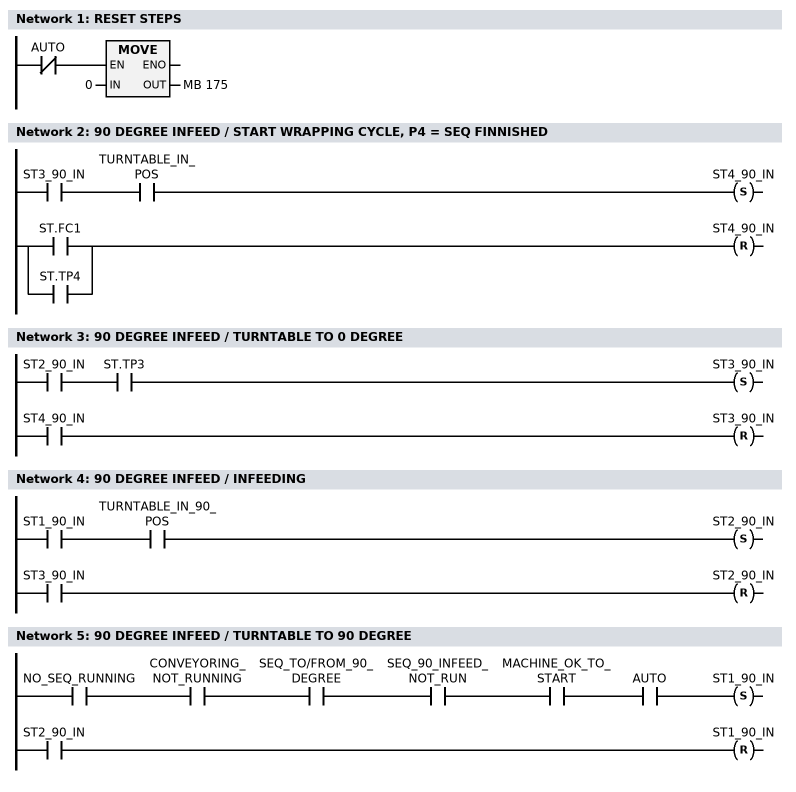
[picture p24: 90_DEGREE_INFEED networks 1-5]
NETWORK
TITLE = RESET STEPS
      AN    "AUTO";
      JNB   _001;
      L     0;
      T     MB 175;
_001: NOP   0;
NETWORK
TITLE = 90 DEGREE INFEED / START WRAPPING CYCLE, P4 = SEQ FINNISHED
      A     "ST3_90_IN";
      A     "TURNTABLE_IN_POS";
      S     "ST4_90_IN";
      A(;
      O     "ST.FC1";
      O     "ST.TP4";
      );
      R     "ST4_90_IN";
      NOP   0;
NETWORK
TITLE = 90 DEGREE INFEED / TURNTABLE TO 0 DEGREE
      A     "ST2_90_IN";
      A     "ST.TP3";
      S     "ST3_90_IN";
      A     "ST4_90_IN";
      R     "ST3_90_IN";
      NOP   0;
NETWORK
TITLE = 90 DEGREE INFEED / INFEEDING
      A     "ST1_90_IN";
      A     "TURNTABLE_IN_90_POS";
      S     "ST2_90_IN";
      A     "ST3_90_IN";
      R     "ST2_90_IN";
      NOP   0;
NETWORK
TITLE = 90 DEGREE INFEED / TURNTABLE TO 90 DEGREE
      A     "NO_SEQ_RUNNING";
      A     "CONVEYORING_NOT_RUNNING";
      A     "SEQ_TO/FROM_90_DEGREE";
      A     "SEQ_90_INFEED_NOT_RUN";
      A     "MACHINE_OK_TO_START";
      A     "AUTO";
      S     "ST1_90_IN";
      A     "ST2_90_IN";
      R     "ST1_90_IN";
      NOP   0;
END_FUNCTION

FUNCTION "90_DEGREE_OUTFEED" : VOID	// FC 18
TITLE = 90 DEGREE OUTFEED, OPTION
AUTHOR : LKA
NAME : OUTF_90D
VERSION : 0.1
BEGIN
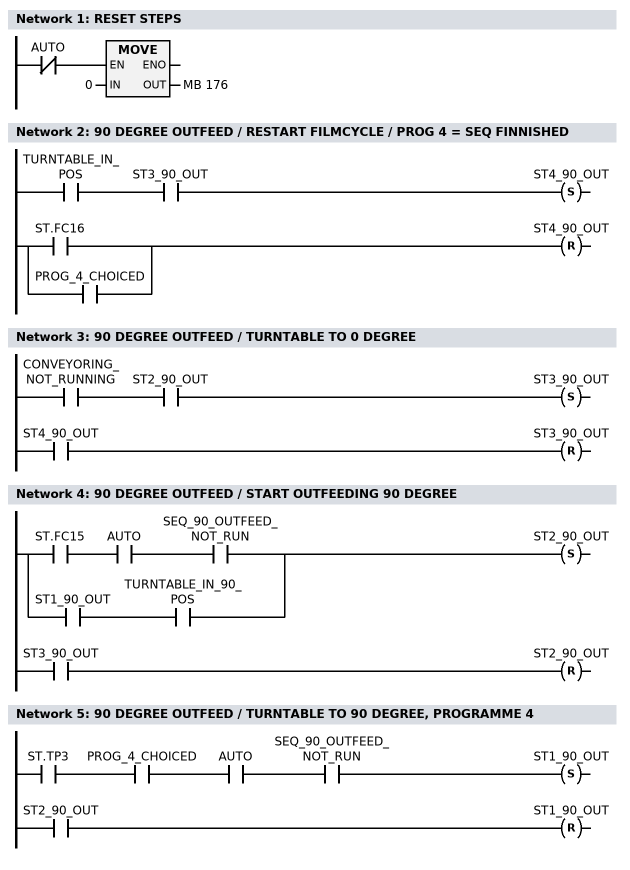
NETWORK
TITLE = RESET STEPS
      AN    "AUTO";
      JNB   _001;
      L     0;
      T     MB 176;
_001: NOP   0;
NETWORK
TITLE = 90 DEGREE OUTFEED / RESTART FILMCYCLE / PROG 4 = SEQ FINNISHED
      A     "TURNTABLE_IN_POS";
      A     "ST3_90_OUT";
      S     "ST4_90_OUT";
      A(;
      O     "ST.FC16";
      O     "PROG_4_CHOICED";
      );
      R     "ST4_90_OUT";
      NOP   0;
NETWORK
TITLE = 90 DEGREE OUTFEED / TURNTABLE TO 0 DEGREE
      A     "CONVEYORING_NOT_RUNNING";
      A     "ST2_90_OUT";
      S     "ST3_90_OUT";
      A     "ST4_90_OUT";
      R     "ST3_90_OUT";
      NOP   0;
NETWORK
TITLE = 90 DEGREE OUTFEED / START OUTFEEDING 90 DEGREE
      A(;
      A     "ST.FC15";
      A     "AUTO";
      A     "SEQ_90_OUTFEED_NOT_RUN";
      O;
      A     "ST1_90_OUT";
      A     "TURNTABLE_IN_90_POS";
      );
      S     "ST2_90_OUT";
      A     "ST3_90_OUT";
      R     "ST2_90_OUT";
      NOP   0;
NETWORK
TITLE = 90 DEGREE OUTFEED / TURNTABLE TO 90 DEGREE, PROGRAMME 4
      A     "ST.TP3";
      A     "PROG_4_CHOICED";
      A     "AUTO";
      A     "SEQ_90_OUTFEED_NOT_RUN";
      S     "ST1_90_OUT";
      A     "ST2_90_OUT";
      R     "ST1_90_OUT";
      NOP   0;
END_FUNCTION

FUNCTION "TURN_TO/FROM_90_DEG" : VOID	// FC 19
TITLE = TURNTABLE TO OR FROM 90 DEGREE, OPTION
AUTHOR : LKA
NAME : TT_90
VERSION : 0.1
BEGIN
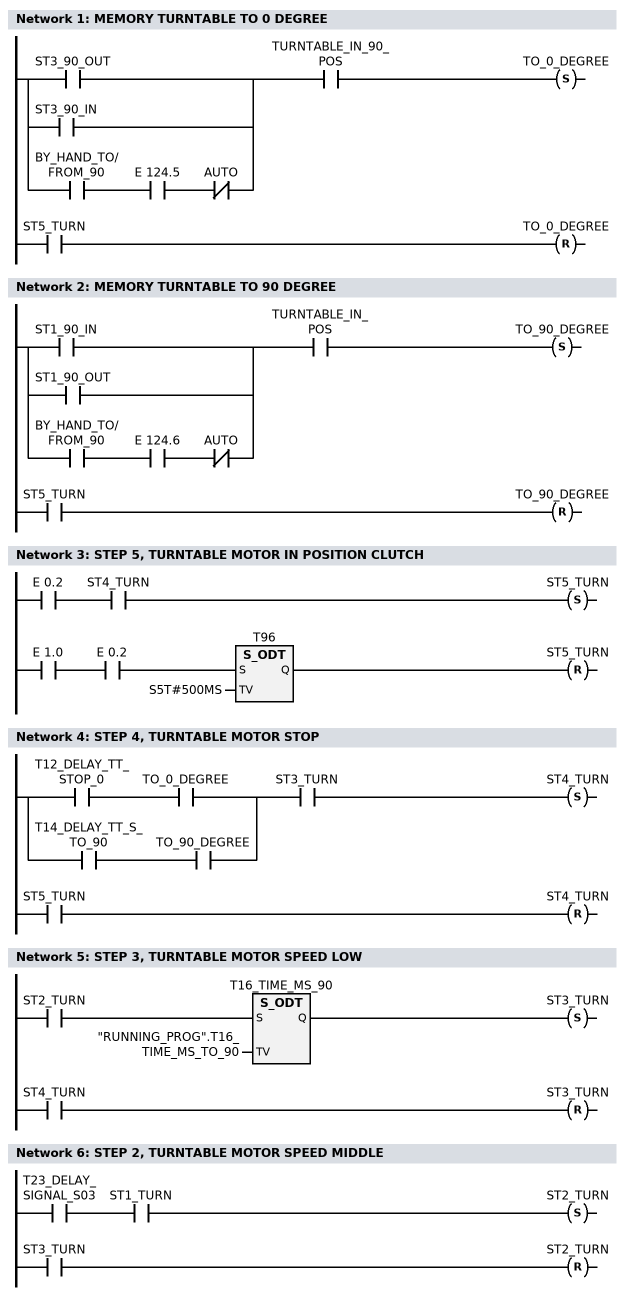
NETWORK
TITLE = MEMORY TURNTABLE TO 0 DEGREE
      A(;
      O     "ST3_90_OUT";
      O     "ST3_90_IN";
      O;
      A     "BY_HAND_TO/FROM_90";
      A     "E 124.5";
      AN    "AUTO";
      );
      A     "TURNTABLE_IN_90_POS";
      S     "TO_0_DEGREE";
      A     "ST5_TURN";
      R     "TO_0_DEGREE";
      NOP   0;
NETWORK
TITLE = MEMORY TURNTABLE TO 90 DEGREE
      A(;
      O     "ST1_90_IN";
      O     "ST1_90_OUT";
      O;
      A     "BY_HAND_TO/FROM_90";
      A     "E 124.6";
      AN    "AUTO";
      );
      A     "TURNTABLE_IN_POS";
      S     "TO_90_DEGREE";
      A     "ST5_TURN";
      R     "TO_90_DEGREE";
      NOP   0;
NETWORK
TITLE = STEP 5, TURNTABLE MOTOR IN POSITION CLUTCH
      A     "E 0.2";
      A     "ST4_TURN";
      S     "ST5_TURN";
      A     "E 1.0";
      A(;
      A     "E 0.2";
      L     S5T#500MS;
      SD    "T96";
      NOP   0;
      NOP   0;
      NOP   0;
      A     "T96";
      );
      R     "ST5_TURN";
      NOP   0;
NETWORK
TITLE = STEP 4, TURNTABLE MOTOR STOP
      A(;
      A     "T12_DELAY_TT_STOP_0";
      A     "TO_0_DEGREE";
      O;
      A     "T14_DELAY_TT_S_TO_90";
      A     "TO_90_DEGREE";
      );
      A     "ST3_TURN";
      S     "ST4_TURN";
      A     "ST5_TURN";
      R     "ST4_TURN";
      NOP   0;
NETWORK
TITLE = STEP 3, TURNTABLE MOTOR SPEED LOW
      A(;
      A     "ST2_TURN";
      L     "RUNNING_PROG".T16_TIME_MS_TO_90;
      SD    "T16_TIME_MS_90";
      NOP   0;
      NOP   0;
      NOP   0;
      A     "T16_TIME_MS_90";
      );
      S     "ST3_TURN";
      A     "ST4_TURN";
      R     "ST3_TURN";
      NOP   0;
NETWORK
TITLE = STEP 2, TURNTABLE MOTOR SPEED MIDDLE
      A     "T23_DELAY_SIGNAL_S03";
      A     "ST1_TURN";
      S     "ST2_TURN";
      A     "ST3_TURN";
      R     "ST2_TURN";
      NOP   0;
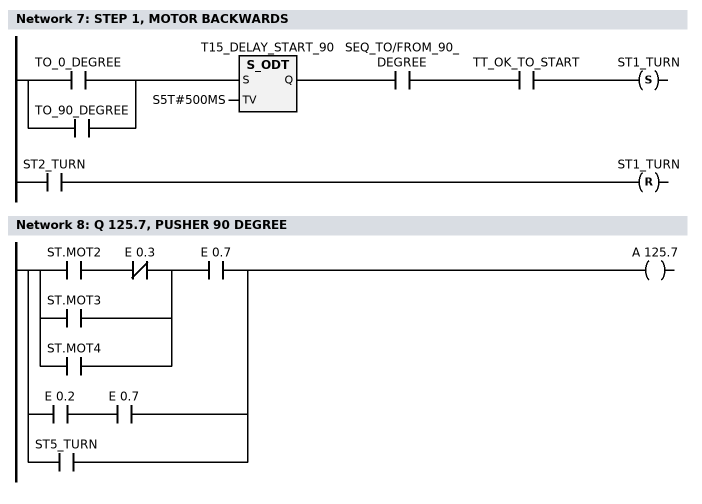
NETWORK
TITLE = STEP 1, MOTOR BACKWARDS
      A(;
      A(;
      O     "TO_0_DEGREE";
      O     "TO_90_DEGREE";
      );
      L     S5T#500MS;
      SD    "T15_DELAY_START_90";
      NOP   0;
      NOP   0;
      NOP   0;
      A     "T15_DELAY_START_90";
      );
      A     "SEQ_TO/FROM_90_DEGREE";
      A     "TT_OK_TO_START";
      S     "ST1_TURN";
      A     "ST2_TURN";
      R     "ST1_TURN";
      NOP   0;
NETWORK
TITLE = Q 125.7, PUSHER 90 DEGREE
      A(;
      A     "ST.MOT2";
      AN    "E 0.3";
      O     "ST.MOT3";
      O     "ST.MOT4";
      );
      A     "E 0.7";
      O;
      A     "E 0.2";
      A     "E 0.7";
      O     "ST5_TURN";
      =     "A 125.7";
END_FUNCTION

FUNCTION "PALLET_POS" : VOID	// FC 21
TITLE = PALLET POSITION - LENGTH MEASURING, OPTION
//OPTIMIZATION OF PALLET STOPTIME ON TURNTABLE
//
//STEP 1: ADJUST CONVEYOR HEIGHT TO BE EQUAL TO STRETCHWRAPPER CONVEYOR, USE A 
//LONG BUBBLE LEVEL.
//
//STEP 2: ADJUST CONVEYOR SPEED ON STRETCHWRAPPER TO BE EQUAL TO INFEEDING 
//CONVEYOR, CHANGE VALUE ON OP3, "TABLEPARAMETERS / CONVEYOR SPEED"
//
//STEP 3: INFEED THE LONGEST PALLET, LOOK AT THE STOP POSITION. ADJUST "Length 
//measuring value" ON OP3 UNTIL THE PALLET STANDS IN MIDDLE. (Counter)
//
//(IF PALLET STOPS TO LATE INCREASE VALUE)
//
//STEP 4: IF NECESSARY, ADJUST OFF DELAY TIME VALUE, T51 & T53 FILTER TIME TO MAKE
//SIGNAL STABLE. (TO LONG TIME MAY CREATE PROBLEM)
AUTHOR : LKA
NAME : L_MATN
VERSION : 1.0
BEGIN
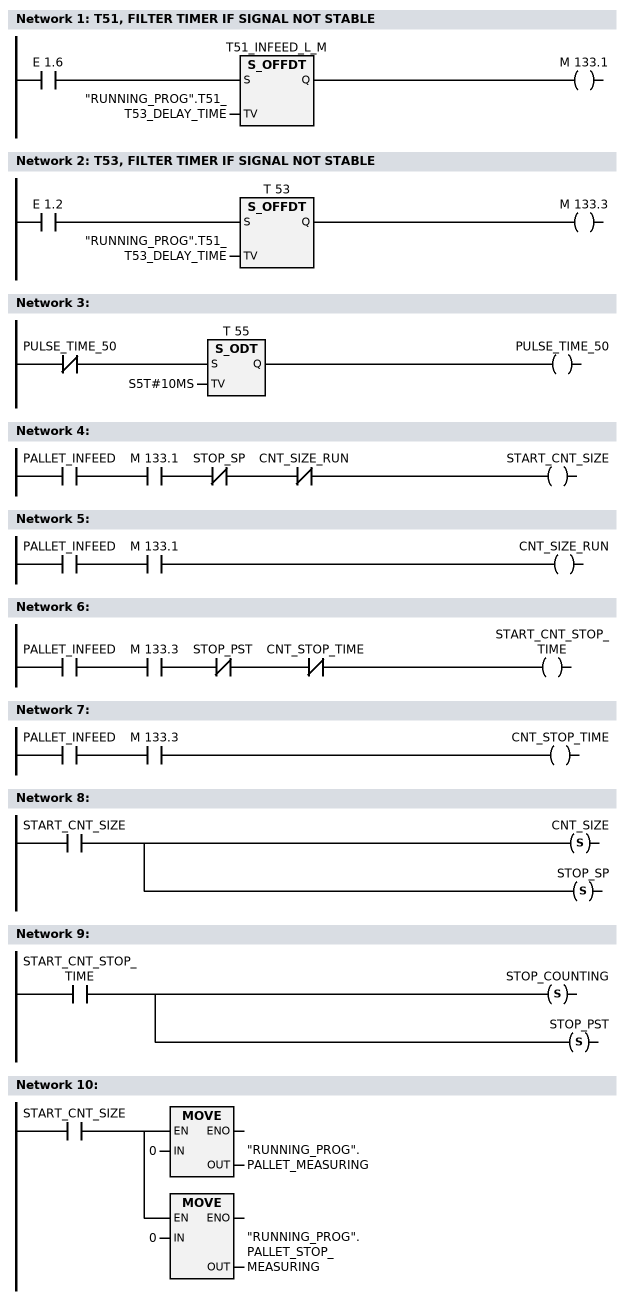
NETWORK
TITLE = T51, FILTER TIMER IF SIGNAL NOT STABLE
      A     "E 1.6";
      L     "RUNNING_PROG".T51_T53_DELAY_TIME;
      SF    "T51_INFEED_L_M";
      NOP   0;
      NOP   0;
      NOP   0;
      A     "T51_INFEED_L_M";
      =     M 133.1;
NETWORK
TITLE = T53, FILTER TIMER IF SIGNAL NOT STABLE
      A     "E 1.2";
      L     "RUNNING_PROG".T51_T53_DELAY_TIME;
      SF    T 53;
      NOP   0;
      NOP   0;
      NOP   0;
      A     T 53;
      =     M 133.3;
NETWORK
TITLE =
      AN    "PULSE_TIME_50";
      L     S5T#10MS;
      SD    T 55;
      NOP   0;
      NOP   0;
      NOP   0;
      A     T 55;
      =     "PULSE_TIME_50";
NETWORK
TITLE =
      A     "PALLET_INFEED";
      A     M 133.1;
      AN    "STOP_SP";
      AN    "CNT_SIZE_RUN";
      =     "START_CNT_SIZE";
NETWORK
TITLE =
      A     "PALLET_INFEED";
      A     M 133.1;
      =     "CNT_SIZE_RUN";
NETWORK
TITLE =
      A     "PALLET_INFEED";
      A     M 133.3;
      AN    "STOP_PST";
      AN    "CNT_STOP_TIME";
      =     "START_CNT_STOP_TIME";
NETWORK
TITLE =
      A     "PALLET_INFEED";
      A     M 133.3;
      =     "CNT_STOP_TIME";
NETWORK
TITLE =
      A     "START_CNT_SIZE";
      S     "CNT_SIZE";
      S     "STOP_SP";
NETWORK
TITLE =
      A     "START_CNT_STOP_TIME";
      S     "STOP_COUNTING";
      S     "STOP_PST";
NETWORK
TITLE =
      A     "START_CNT_SIZE";
      =     L 172.0;
      A     L 172.0;
      JNB   _001;
      L     0;
      T     "RUNNING_PROG".PALLET_MEASURING;
_001: NOP   0;
      A     L 172.0;
      JNB   _002;
      L     0;
      T     "RUNNING_PROG".PALLET_STOP_MEASURING;
_002: NOP   0;
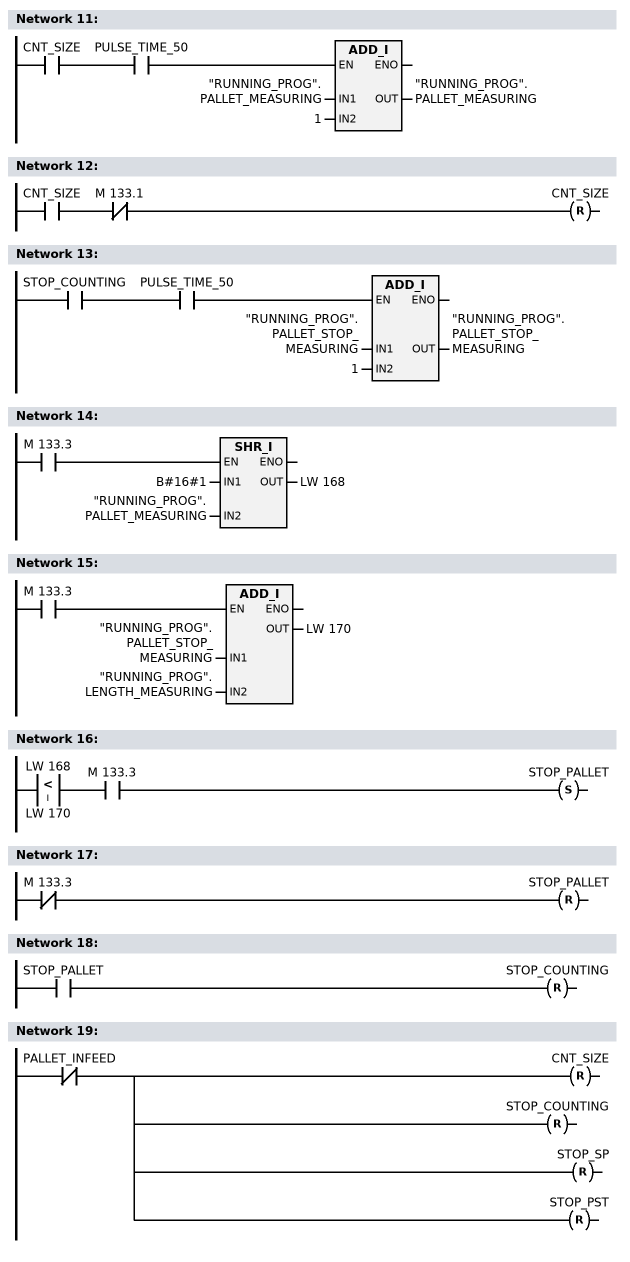
NETWORK
TITLE =
      A     "CNT_SIZE";
      A     "PULSE_TIME_50";
      JNB   _003;
      L     "RUNNING_PROG".PALLET_MEASURING;
      L     1;
      +I;
      T     "RUNNING_PROG".PALLET_MEASURING;
_003: NOP   0;
NETWORK
TITLE =
      A     "CNT_SIZE";
      AN    M 133.1;
      R     "CNT_SIZE";
NETWORK
TITLE =
      A     "STOP_COUNTING";
      A     "PULSE_TIME_50";
      JNB   _004;
      L     "RUNNING_PROG".PALLET_STOP_MEASURING;
      L     1;
      +I;
      T     "RUNNING_PROG".PALLET_STOP_MEASURING;
_004: NOP   0;
NETWORK
TITLE =
      A     M 133.3;
      JNB   _005;
      L     B#16#1;
      L     "RUNNING_PROG".PALLET_MEASURING;
      SSI;
      T     LW 168;
_005: NOP   0;
NETWORK
TITLE =
      A     M 133.3;
      JNB   _006;
      L     "RUNNING_PROG".PALLET_STOP_MEASURING;
      L     "RUNNING_PROG".LENGTH_MEASURING;
      +I;
      T     LW 170;
_006: NOP   0;
NETWORK
TITLE =
      A(;
      L     LW 168;
      L     LW 170;
      <I;
      );
      A     M 133.3;
      S     "STOP_PALLET";
NETWORK
TITLE =
      AN    M 133.3;
      R     "STOP_PALLET";
NETWORK
TITLE =
      A     "STOP_PALLET";
      R     "STOP_COUNTING";
NETWORK
TITLE =
      AN    "PALLET_INFEED";
      R     "CNT_SIZE";
      R     "STOP_COUNTING";
      R     "STOP_SP";
      R     "STOP_PST";
END_FUNCTION

FUNCTION "TURNTABLE" : VOID	// FC 22
TITLE = TURNTABLE
AUTHOR : LKA
NAME : TURNTAB
VERSION : 0.0
BEGIN
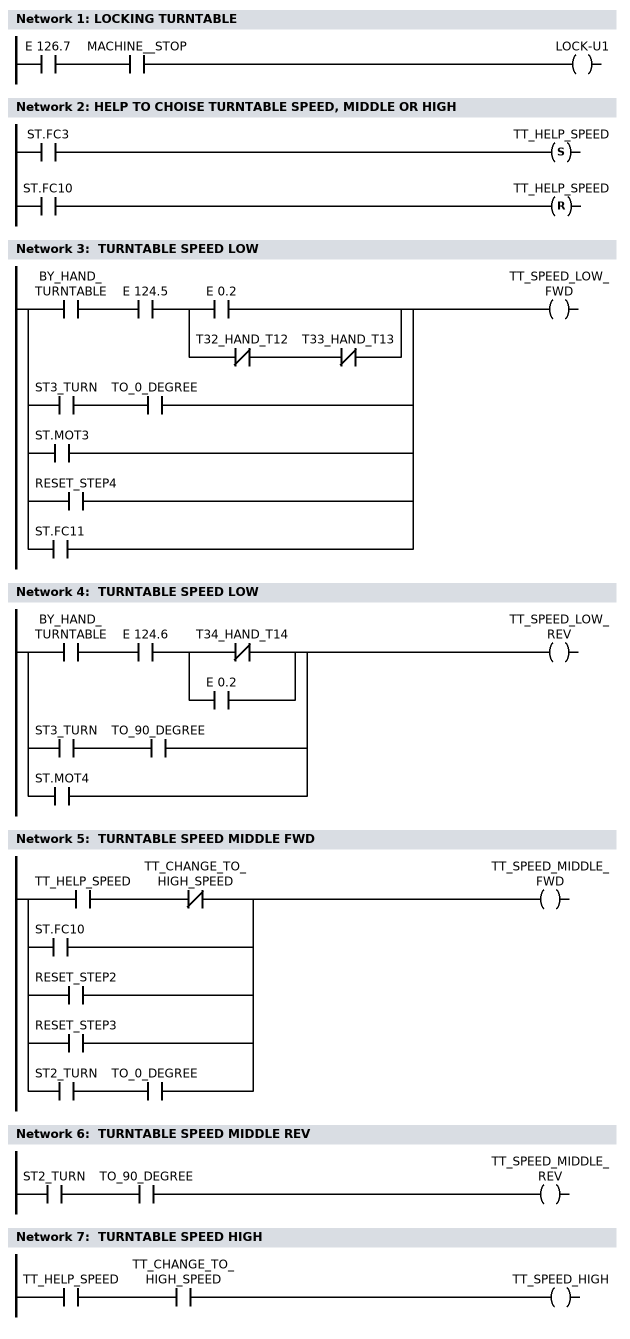
NETWORK
TITLE = LOCKING TURNTABLE
      A     "E 126.7";
      A     "MACHINE__STOP";
      =     "LOCK-U1";
NETWORK
TITLE = HELP TO CHOISE TURNTABLE SPEED, MIDDLE OR HIGH
      A     "ST.FC3";
      S     "TT_HELP_SPEED";
      A     "ST.FC10";
      R     "TT_HELP_SPEED";
      NOP   0;
NETWORK
TITLE =  TURNTABLE SPEED LOW
      A     "BY_HAND_TURNTABLE";
      A     "E 124.5";
      A(;
      O     "E 0.2";
      O;
      AN    "T32_HAND_T12";
      AN    "T33_HAND_T13";
      );
      O;
      A     "ST3_TURN";
      A     "TO_0_DEGREE";
      O     "ST.MOT3";
      O     "RESET_STEP4";
      O     "ST.FC11";
      =     "TT_SPEED_LOW_FWD";
NETWORK
TITLE =  TURNTABLE SPEED LOW
      A     "BY_HAND_TURNTABLE";
      A     "E 124.6";
      A(;
      ON    "T34_HAND_T14";
      O     "E 0.2";
      );
      O;
      A     "ST3_TURN";
      A     "TO_90_DEGREE";
      O     "ST.MOT4";
      =     "TT_SPEED_LOW_REV";
NETWORK
TITLE =  TURNTABLE SPEED MIDDLE FWD
      A     "TT_HELP_SPEED";
      AN    "TT_CHANGE_TO_HIGH_SPEED";
      O     "ST.FC10";
      O     "RESET_STEP2";
      O     "RESET_STEP3";
      O;
      A     "ST2_TURN";
      A     "TO_0_DEGREE";
      =     "TT_SPEED_MIDDLE_FWD";
NETWORK
TITLE =  TURNTABLE SPEED MIDDLE REV
      A     "ST2_TURN";
      A     "TO_90_DEGREE";
      =     "TT_SPEED_MIDDLE_REV";
NETWORK
TITLE =  TURNTABLE SPEED HIGH
      A     "TT_HELP_SPEED";
      A     "TT_CHANGE_TO_HIGH_SPEED";
      =     "TT_SPEED_HIGH";
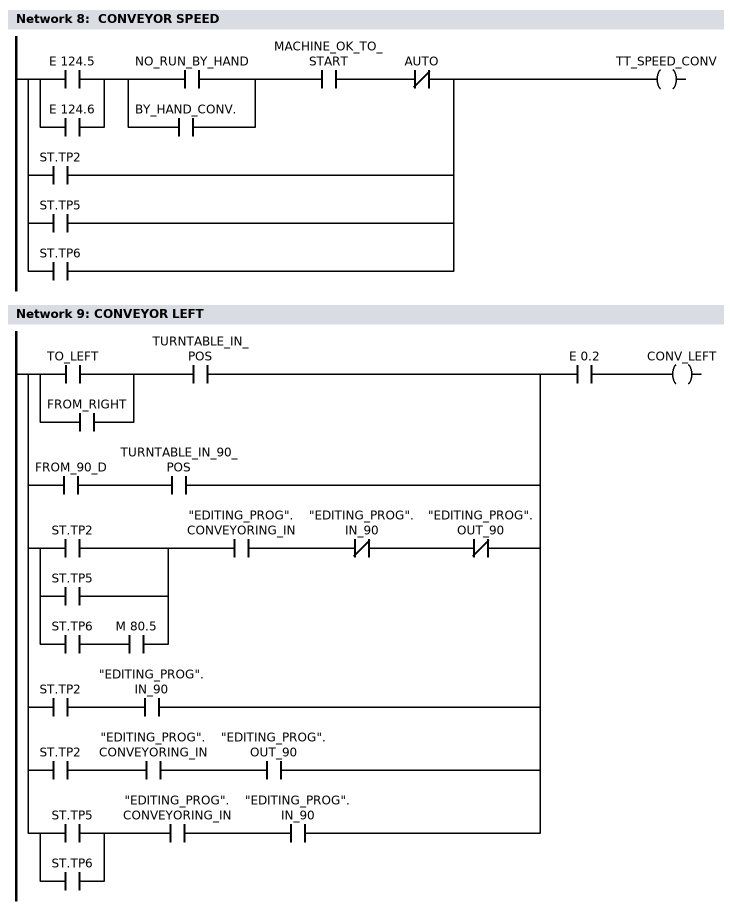
NETWORK
TITLE =  CONVEYOR SPEED
      A(;
      O     "E 124.5";
      O     "E 124.6";
      );
      A(;
      O     "NO_RUN_BY_HAND";
      O     "BY_HAND_CONV.";
      );
      A     "MACHINE_OK_TO_START";
      AN    "AUTO";
      O     "ST.TP2";
      O     "ST.TP5";
      O     "ST.TP6";
      =     "TT_SPEED_CONV";
NETWORK
TITLE = CONVEYOR LEFT
      A(;
      A(;
      O     "TO_LEFT";
      O     "FROM_RIGHT";
      );
      A     "TURNTABLE_IN_POS";
      O;
      A     "FROM_90_D";
      A     "TURNTABLE_IN_90_POS";
      O;
      A(;
      O     "ST.TP2";
      O     "ST.TP5";
      O;
      A     "ST.TP6";
      A     "M 80.5";
      );
      A     "EDITING_PROG".CONVEYORING_IN;
      AN    "EDITING_PROG".IN_90;
      AN    "EDITING_PROG".OUT_90;
      O;
      A     "ST.TP2";
      A     "EDITING_PROG".IN_90;
      O;
      A     "ST.TP2";
      A     "EDITING_PROG".CONVEYORING_IN;
      A     "EDITING_PROG".OUT_90;
      O;
      A(;
      O     "ST.TP5";
      O     "ST.TP6";
      );
      A     "EDITING_PROG".CONVEYORING_IN;
      A     "EDITING_PROG".IN_90;
      );
      A     "E 0.2";
      =     "CONV_LEFT";
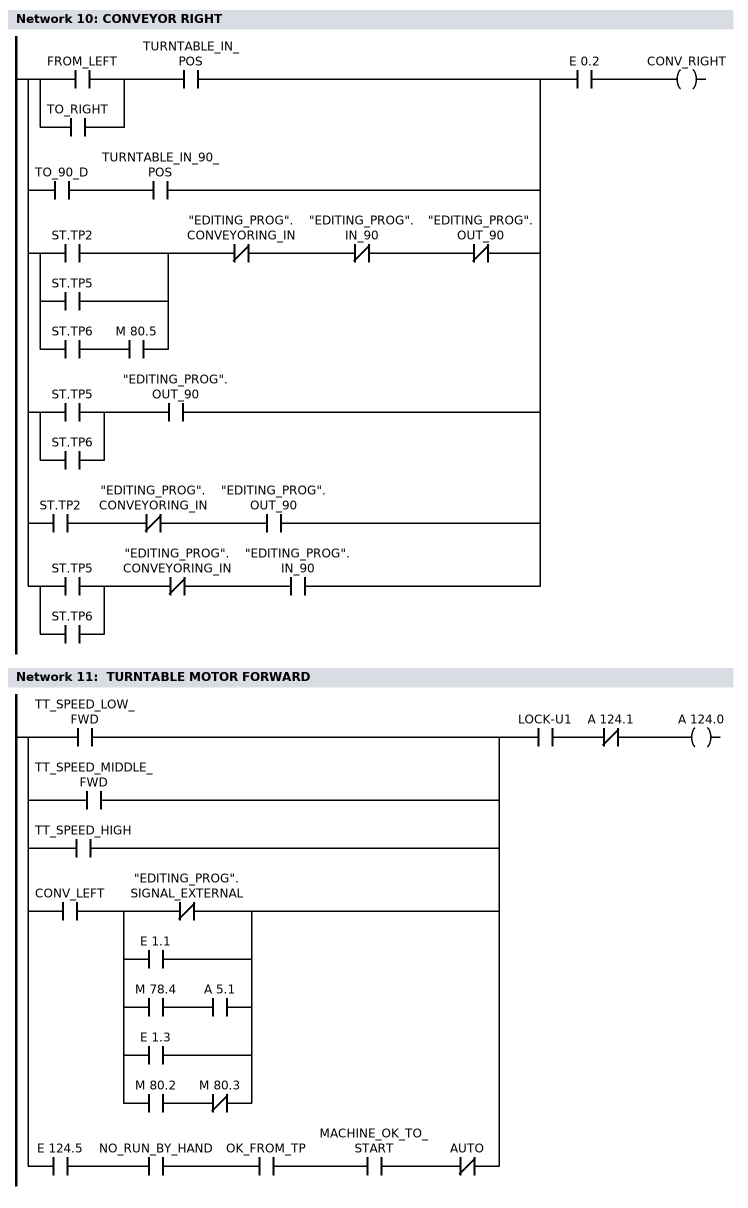
NETWORK
TITLE = CONVEYOR RIGHT
      A(;
      A(;
      O     "FROM_LEFT";
      O     "TO_RIGHT";
      );
      A     "TURNTABLE_IN_POS";
      O;
      A     "TO_90_D";
      A     "TURNTABLE_IN_90_POS";
      O;
      A(;
      O     "ST.TP2";
      O     "ST.TP5";
      O;
      A     "ST.TP6";
      A     "M 80.5";
      );
      AN    "EDITING_PROG".CONVEYORING_IN;
      AN    "EDITING_PROG".IN_90;
      AN    "EDITING_PROG".OUT_90;
      O;
      A(;
      O     "ST.TP5";
      O     "ST.TP6";
      );
      A     "EDITING_PROG".OUT_90;
      O;
      A     "ST.TP2";
      AN    "EDITING_PROG".CONVEYORING_IN;
      A     "EDITING_PROG".OUT_90;
      O;
      A(;
      O     "ST.TP5";
      O     "ST.TP6";
      );
      AN    "EDITING_PROG".CONVEYORING_IN;
      A     "EDITING_PROG".IN_90;
      );
      A     "E 0.2";
      =     "CONV_RIGHT";
NETWORK
TITLE =  TURNTABLE MOTOR FORWARD
      A(;
      O     "TT_SPEED_LOW_FWD";
      O     "TT_SPEED_MIDDLE_FWD";
      O     "TT_SPEED_HIGH";
      O;
      A     "CONV_LEFT";
      A(;
      ON    "EDITING_PROG".SIGNAL_EXTERNAL;
      O     "E 1.1";
      O;
      A     "M 78.4";
      A     "A 5.1";
      O     "E 1.3";
      O;
      A     "M 80.2";
      AN    "M 80.3";
      );
      O;
      A     "E 124.5";
      A     "NO_RUN_BY_HAND";
      A     "OK_FROM_TP";
      A     "MACHINE_OK_TO_START";
      AN    "AUTO";
      );
      A     "LOCK-U1";
      AN    "A 124.1";
      =     "A 124.0";
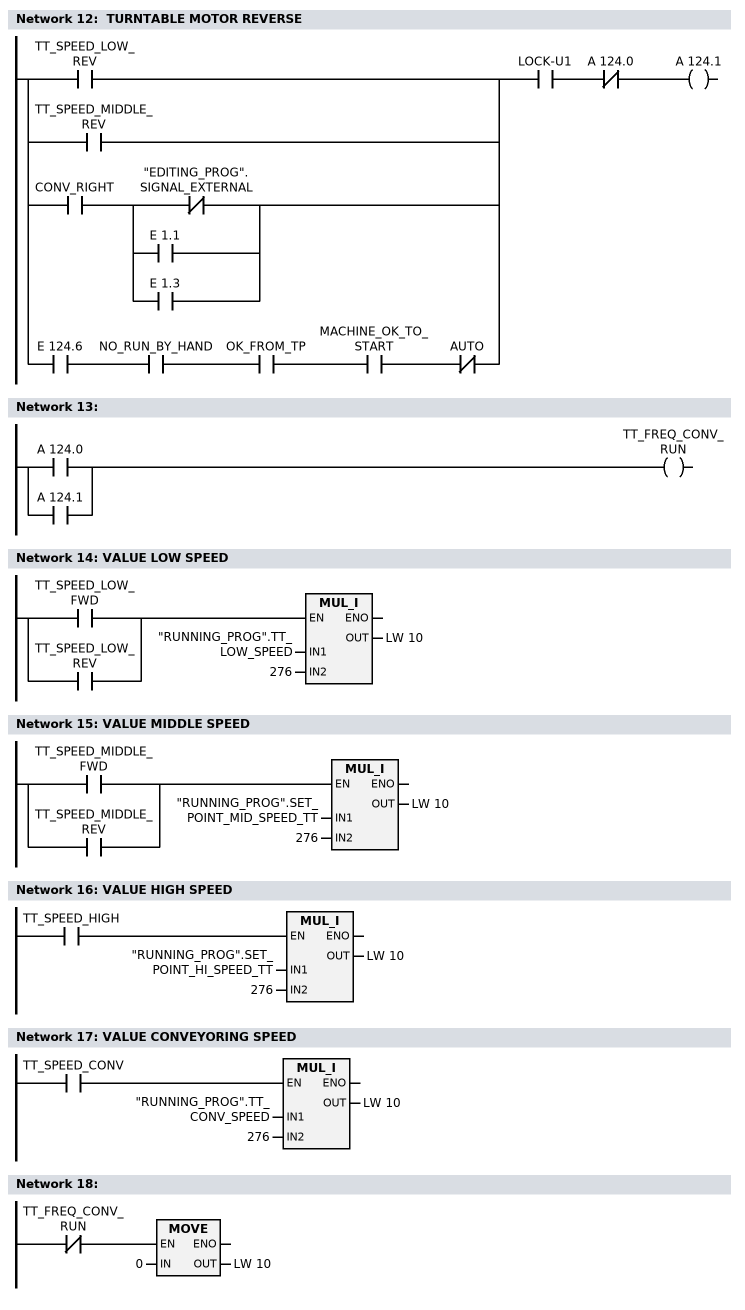
NETWORK
TITLE =  TURNTABLE MOTOR REVERSE
      A(;
      O     "TT_SPEED_LOW_REV";
      O     "TT_SPEED_MIDDLE_REV";
      O;
      A     "CONV_RIGHT";
      A(;
      ON    "EDITING_PROG".SIGNAL_EXTERNAL;
      O     "E 1.1";
      O     "E 1.3";
      );
      O;
      A     "E 124.6";
      A     "NO_RUN_BY_HAND";
      A     "OK_FROM_TP";
      A     "MACHINE_OK_TO_START";
      AN    "AUTO";
      );
      A     "LOCK-U1";
      AN    "A 124.0";
      =     "A 124.1";
NETWORK
TITLE =
      O     "A 124.0";
      O     "A 124.1";
      =     "TT_FREQ_CONV_RUN";
NETWORK
TITLE = VALUE LOW SPEED
      A(;
      O     "TT_SPEED_LOW_FWD";
      O     "TT_SPEED_LOW_REV";
      );
      JNB   _001;
      L     "RUNNING_PROG".TT_LOW_SPEED;
      L     276;
      *I;
      T     LW 10;
_001: NOP   0;
NETWORK
TITLE = VALUE MIDDLE SPEED
      A(;
      O     "TT_SPEED_MIDDLE_FWD";
      O     "TT_SPEED_MIDDLE_REV";
      );
      JNB   _002;
      L     "RUNNING_PROG".SET_POINT_MID_SPEED_TT;
      L     276;
      *I;
      T     LW 10;
_002: NOP   0;
NETWORK
TITLE = VALUE HIGH SPEED
      A     "TT_SPEED_HIGH";
      JNB   _003;
      L     "RUNNING_PROG".SET_POINT_HI_SPEED_TT;
      L     276;
      *I;
      T     LW 10;
_003: NOP   0;
NETWORK
TITLE = VALUE CONVEYORING SPEED
      A     "TT_SPEED_CONV";
      JNB   _004;
      L     "RUNNING_PROG".TT_CONV_SPEED;
      L     276;
      *I;
      T     LW 10;
_004: NOP   0;
NETWORK
TITLE =
      AN    "TT_FREQ_CONV_RUN";
      JNB   _005;
      L     0;
      T     LW 10;
_005: NOP   0;
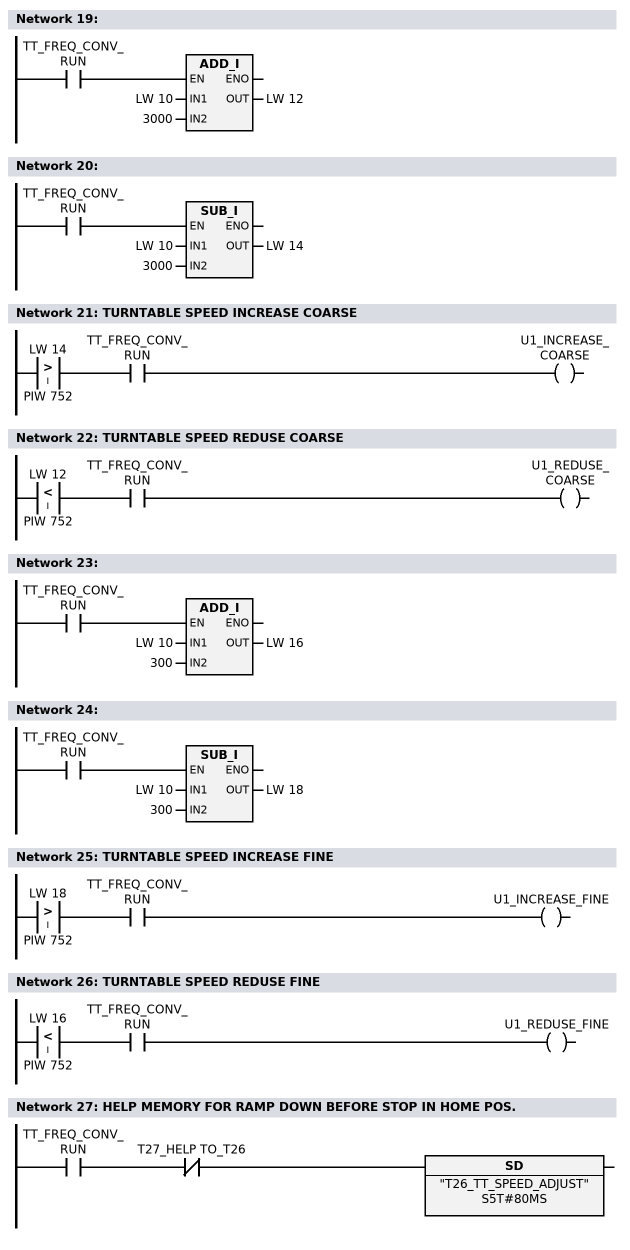
NETWORK
TITLE =
      A     "TT_FREQ_CONV_RUN";
      JNB   _006;
      L     LW 10;
      L     3000;
      +I;
      T     LW 12;
_006: NOP   0;
NETWORK
TITLE =
      A     "TT_FREQ_CONV_RUN";
      JNB   _007;
      L     LW 10;
      L     3000;
      -I;
      T     LW 14;
_007: NOP   0;
NETWORK
TITLE = TURNTABLE SPEED INCREASE COARSE
      A(;
      L     LW 14;
      L     PIW 752;
      >I;
      );
      A     "TT_FREQ_CONV_RUN";
      =     "U1_INCREASE_COARSE";
NETWORK
TITLE = TURNTABLE SPEED REDUSE COARSE
      A(;
      L     LW 12;
      L     PIW 752;
      <I;
      );
      A     "TT_FREQ_CONV_RUN";
      =     "U1_REDUSE_COARSE";
NETWORK
TITLE =
      A     "TT_FREQ_CONV_RUN";
      JNB   _008;
      L     LW 10;
      L     300;
      +I;
      T     LW 16;
_008: NOP   0;
NETWORK
TITLE =
      A     "TT_FREQ_CONV_RUN";
      JNB   _009;
      L     LW 10;
      L     300;
      -I;
      T     LW 18;
_009: NOP   0;
NETWORK
TITLE = TURNTABLE SPEED INCREASE FINE
      A(;
      L     LW 18;
      L     PIW 752;
      >I;
      );
      A     "TT_FREQ_CONV_RUN";
      =     "U1_INCREASE_FINE";
NETWORK
TITLE = TURNTABLE SPEED REDUSE FINE
      A(;
      L     LW 16;
      L     PIW 752;
      <I;
      );
      A     "TT_FREQ_CONV_RUN";
      =     "U1_REDUSE_FINE";
NETWORK
TITLE = HELP MEMORY FOR RAMP DOWN BEFORE STOP IN HOME POS.
      A     "TT_FREQ_CONV_RUN";
      AN    "T27_HELP TO_T26";
      L     S5T#80MS;
      SD    "T26_TT_SPEED_ADJUST";
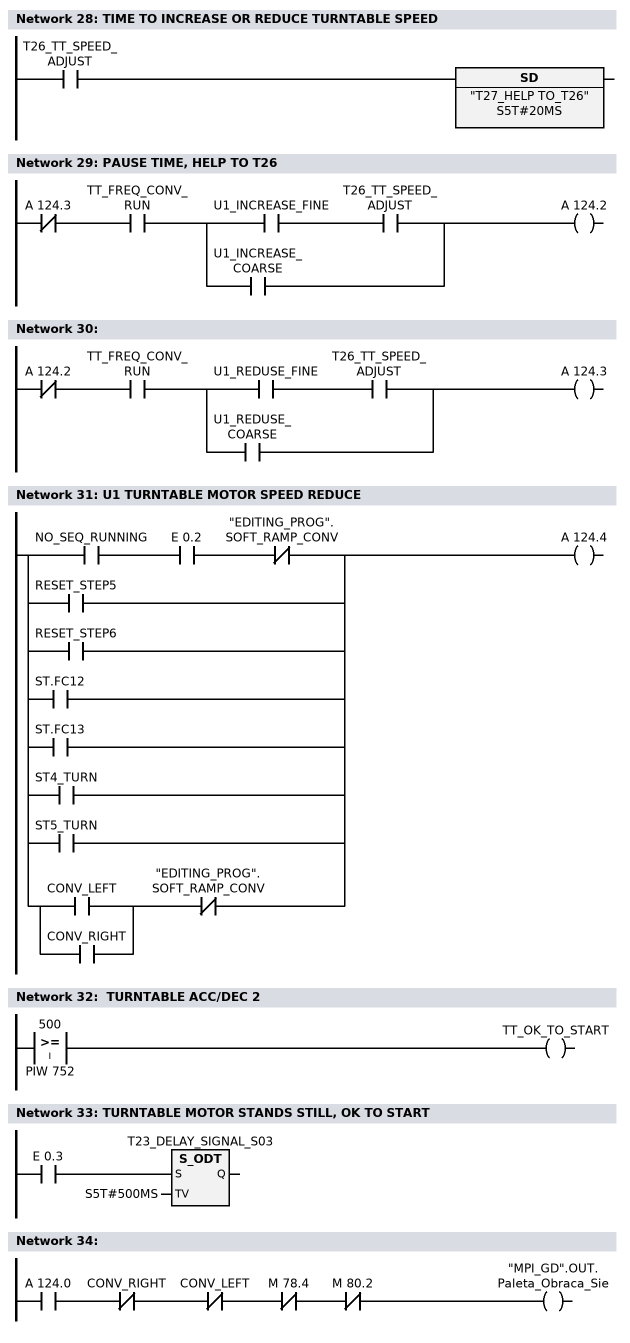
NETWORK
TITLE = TIME TO INCREASE OR REDUCE TURNTABLE SPEED
      A     "T26_TT_SPEED_ADJUST";
      L     S5T#20MS;
      SD    "T27_HELP TO_T26";
NETWORK
TITLE = PAUSE TIME, HELP TO T26
      AN    "A 124.3";
      A     "TT_FREQ_CONV_RUN";
      A(;
      A     "U1_INCREASE_FINE";
      A     "T26_TT_SPEED_ADJUST";
      O     "U1_INCREASE_COARSE";
      );
      =     "A 124.2";
NETWORK
TITLE =
      AN    "A 124.2";
      A     "TT_FREQ_CONV_RUN";
      A(;
      A     "U1_REDUSE_FINE";
      A     "T26_TT_SPEED_ADJUST";
      O     "U1_REDUSE_COARSE";
      );
      =     "A 124.3";
NETWORK
TITLE = U1 TURNTABLE MOTOR SPEED REDUCE
      A     "NO_SEQ_RUNNING";
      A     "E 0.2";
      AN    "EDITING_PROG".SOFT_RAMP_CONV;
      O     "RESET_STEP5";
      O     "RESET_STEP6";
      O     "ST.FC12";
      O     "ST.FC13";
      O     "ST4_TURN";
      O     "ST5_TURN";
      O;
      A(;
      O     "CONV_LEFT";
      O     "CONV_RIGHT";
      );
      AN    "EDITING_PROG".SOFT_RAMP_CONV;
      =     "A 124.4";
NETWORK
TITLE =  TURNTABLE ACC/DEC 2
//skall kollas!!!! ev S/R för trp, inte bordsmotor = reset (&n fwd+rev)
      L     500;
      L     PIW 752;
      >=I;
      =     "TT_OK_TO_START";
NETWORK
TITLE = TURNTABLE MOTOR STANDS STILL, OK TO START
      A     "E 0.3";
      L     S5T#500MS;
      SD    "T23_DELAY_SIGNAL_S03";
      NOP   0;
      NOP   0;
      NOP   0;
      NOP   0;
NETWORK
TITLE =
      A     "A 124.0";
      AN    "CONV_RIGHT";
      AN    "CONV_LEFT";
      AN    "M 78.4";
      AN    "M 80.2";
      =     "MPI_GD".OUT.Paleta_Obraca_Sie;
END_FUNCTION

FUNCTION "CARRIAGE" : VOID	// FC 23
TITLE = CARRIAGE
AUTHOR : LKA
NAME : CARR
VERSION : 0.0
BEGIN
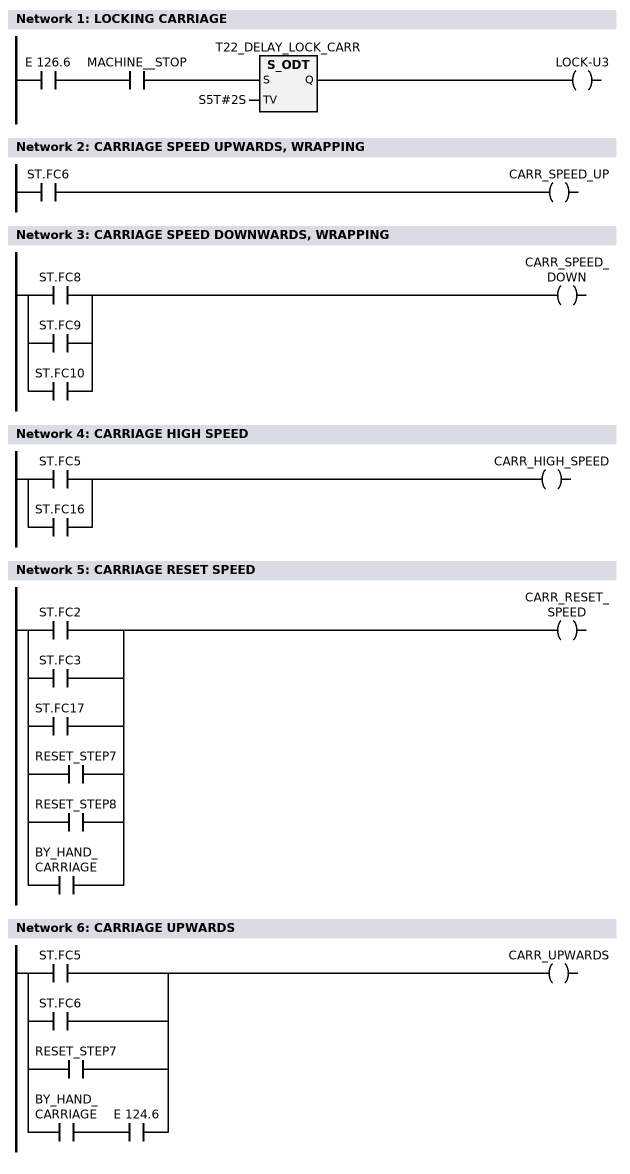
NETWORK
TITLE = LOCKING CARRIAGE
//BÖR HA EJ TILLSLAGS FÖRDRÖJD TID FFÖR ATT HÅLLA HISS EFTER MASKIN STOPP.
      A     "E 126.6";
      A     "MACHINE__STOP";
      L     S5T#2S;
      SD    "T22_DELAY_LOCK_CARR";
      NOP   0;
      NOP   0;
      NOP   0;
      A     "T22_DELAY_LOCK_CARR";
      =     "LOCK-U3";
NETWORK
TITLE = CARRIAGE SPEED UPWARDS, WRAPPING
      A     "ST.FC6";
      =     "CARR_SPEED_UP";
NETWORK
TITLE = CARRIAGE SPEED DOWNWARDS, WRAPPING
      O     "ST.FC8";
      O     "ST.FC9";
      O     "ST.FC10";
      =     "CARR_SPEED_DOWN";
NETWORK
TITLE = CARRIAGE HIGH SPEED
      O     "ST.FC5";
      O     "ST.FC16";
      =     "CARR_HIGH_SPEED";
NETWORK
TITLE = CARRIAGE RESET SPEED
      O     "ST.FC2";
      O     "ST.FC3";
      O     "ST.FC17";
      O     "RESET_STEP7";
      O     "RESET_STEP8";
      O     "BY_HAND_CARRIAGE";
      =     "CARR_RESET_SPEED";
NETWORK
TITLE = CARRIAGE UPWARDS
//MINSTA HÖJD??
      O     "ST.FC5";
      O     "ST.FC6";
      O     "RESET_STEP7";
      O;
      A     "BY_HAND_CARRIAGE";
      A     "E 124.6";
      =     "CARR_UPWARDS";
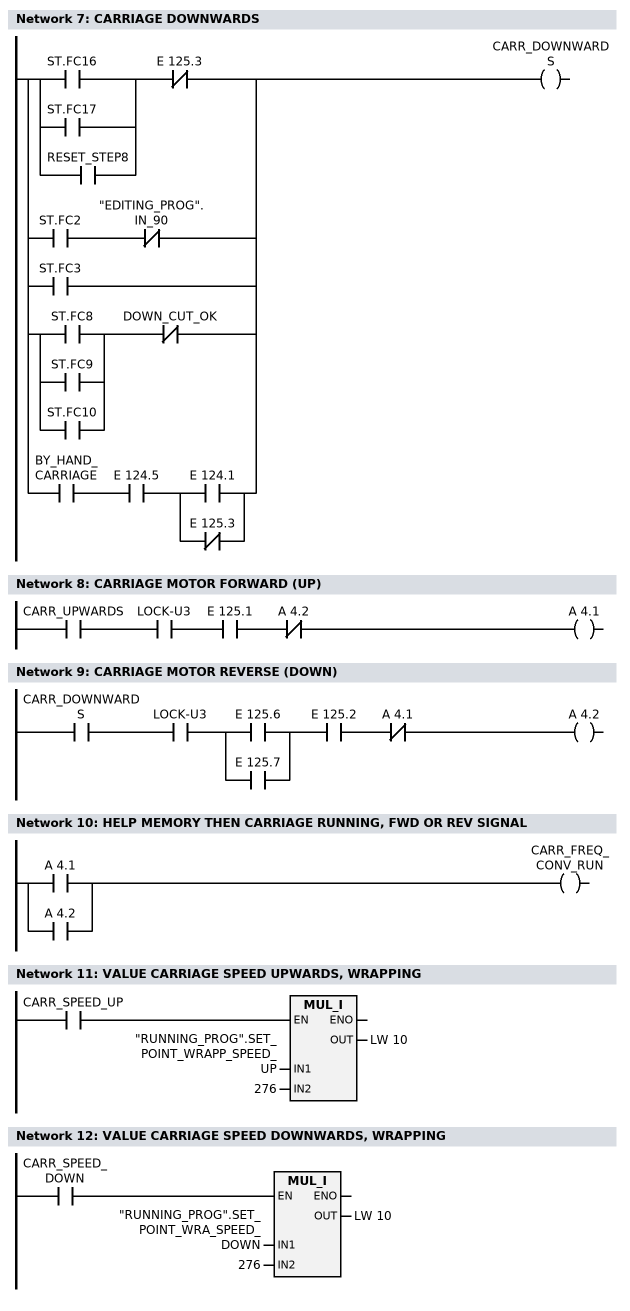
NETWORK
TITLE = CARRIAGE DOWNWARDS
//MINSTA HÖJD????
      A(;
      O     "ST.FC16";
      O     "ST.FC17";
      O     "RESET_STEP8";
      );
      AN    "E 125.3";
      O;
      A     "ST.FC2";
      AN    "EDITING_PROG".IN_90;
      O     "ST.FC3";
      O;
      A(;
      O     "ST.FC8";
      O     "ST.FC9";
      O     "ST.FC10";
      );
      AN    "DOWN_CUT_OK";
      O;
      A     "BY_HAND_CARRIAGE";
      A     "E 124.5";
      A(;
      O     "E 124.1";
      ON    "E 125.3";
      );
      =     "CARR_DOWNWARDS";
NETWORK
TITLE = CARRIAGE MOTOR FORWARD (UP)
//KOLLAS!!
      A     "CARR_UPWARDS";
      A     "LOCK-U3";
      A     "E 125.1";
      AN    "A 4.2";
      =     "A 4.1";
NETWORK
TITLE = CARRIAGE MOTOR REVERSE (DOWN)
//koLLAS!!
      A     "CARR_DOWNWARDS";
      A     "LOCK-U3";
      A(;
      O     "E 125.6";
      O     "E 125.7";
      );
      A     "E 125.2";
      AN    "A 4.1";
      =     "A 4.2";
NETWORK
TITLE = HELP MEMORY THEN CARRIAGE RUNNING, FWD OR REV SIGNAL
      O     "A 4.1";
      O     "A 4.2";
      =     "CARR_FREQ_CONV_RUN";
NETWORK
TITLE = VALUE CARRIAGE SPEED UPWARDS, WRAPPING
      A     "CARR_SPEED_UP";
      JNB   _001;
      L     "RUNNING_PROG".SET_POINT_WRAPP_SPEED_UP;
      L     276;
      *I;
      T     LW 10;
_001: NOP   0;
NETWORK
TITLE = VALUE CARRIAGE SPEED DOWNWARDS, WRAPPING
      A     "CARR_SPEED_DOWN";
      JNB   _002;
      L     "RUNNING_PROG".SET_POINT_WRA_SPEED_DOWN;
      L     276;
      *I;
      T     LW 10;
_002: NOP   0;
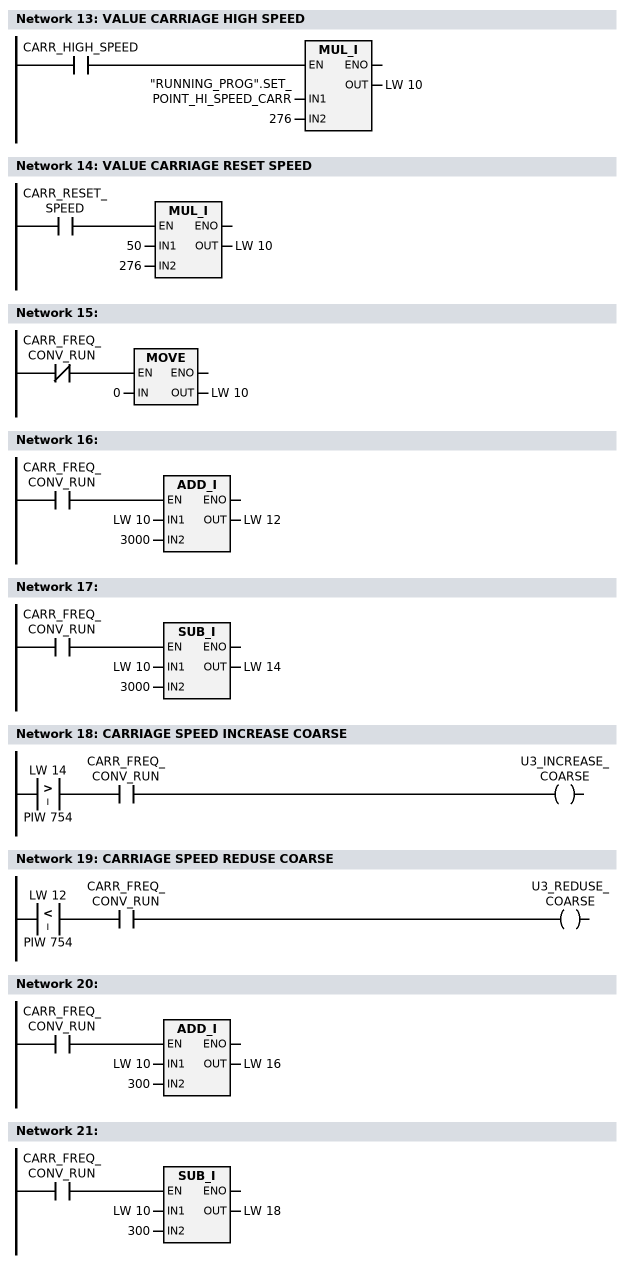
NETWORK
TITLE = VALUE CARRIAGE HIGH SPEED
      A     "CARR_HIGH_SPEED";
      JNB   _003;
      L     "RUNNING_PROG".SET_POINT_HI_SPEED_CARR;
      L     276;
      *I;
      T     LW 10;
_003: NOP   0;
NETWORK
TITLE = VALUE CARRIAGE RESET SPEED
      A     "CARR_RESET_SPEED";
      JNB   _004;
      L     50;
      L     276;
      *I;
      T     LW 10;
_004: NOP   0;
NETWORK
TITLE =
      AN    "CARR_FREQ_CONV_RUN";
      JNB   _005;
      L     0;
      T     LW 10;
_005: NOP   0;
NETWORK
TITLE =
      A     "CARR_FREQ_CONV_RUN";
      JNB   _006;
      L     LW 10;
      L     3000;
      +I;
      T     LW 12;
_006: NOP   0;
NETWORK
TITLE =
      A     "CARR_FREQ_CONV_RUN";
      JNB   _007;
      L     LW 10;
      L     3000;
      -I;
      T     LW 14;
_007: NOP   0;
NETWORK
TITLE = CARRIAGE SPEED INCREASE COARSE
      A(;
      L     LW 14;
      L     PIW 754;
      >I;
      );
      A     "CARR_FREQ_CONV_RUN";
      =     "U3_INCREASE_COARSE";
NETWORK
TITLE = CARRIAGE SPEED REDUSE COARSE
      A(;
      L     LW 12;
      L     PIW 754;
      <I;
      );
      A     "CARR_FREQ_CONV_RUN";
      =     "U3_REDUSE_COARSE";
NETWORK
TITLE =
      A     "CARR_FREQ_CONV_RUN";
      JNB   _008;
      L     LW 10;
      L     300;
      +I;
      T     LW 16;
_008: NOP   0;
NETWORK
TITLE =
      A     "CARR_FREQ_CONV_RUN";
      JNB   _009;
      L     LW 10;
      L     300;
      -I;
      T     LW 18;
_009: NOP   0;
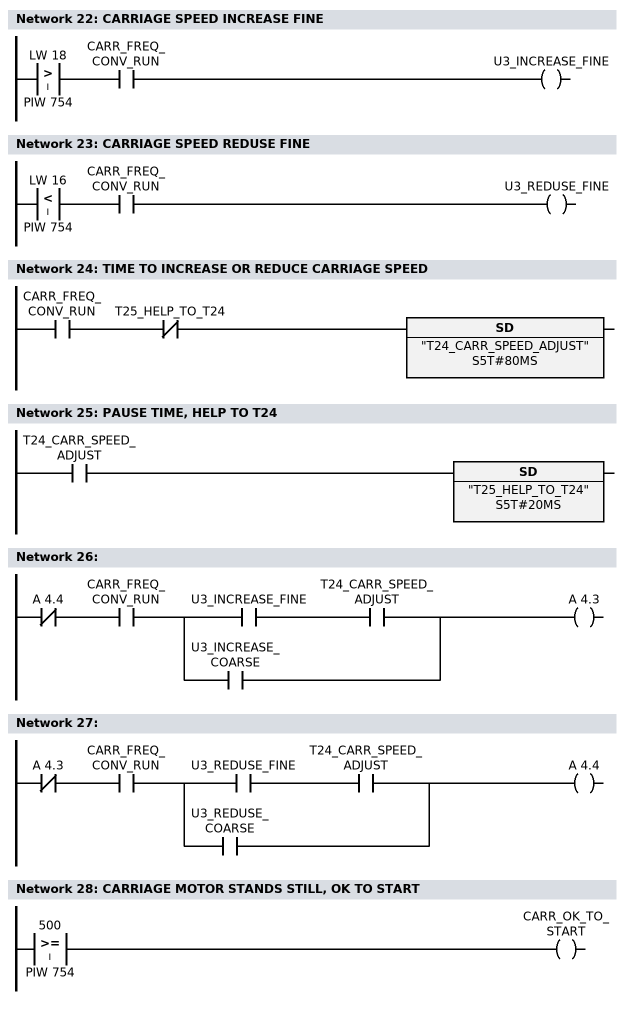
NETWORK
TITLE = CARRIAGE SPEED INCREASE FINE
      A(;
      L     LW 18;
      L     PIW 754;
      >I;
      );
      A     "CARR_FREQ_CONV_RUN";
      =     "U3_INCREASE_FINE";
NETWORK
TITLE = CARRIAGE SPEED REDUSE FINE
      A(;
      L     LW 16;
      L     PIW 754;
      <I;
      );
      A     "CARR_FREQ_CONV_RUN";
      =     "U3_REDUSE_FINE";
NETWORK
TITLE = TIME TO INCREASE OR REDUCE CARRIAGE SPEED
      A     "CARR_FREQ_CONV_RUN";
      AN    "T25_HELP_TO_T24";
      L     S5T#80MS;
      SD    "T24_CARR_SPEED_ADJUST";
NETWORK
TITLE = PAUSE TIME, HELP TO T24
      A     "T24_CARR_SPEED_ADJUST";
      L     S5T#20MS;
      SD    "T25_HELP_TO_T24";
NETWORK
TITLE =
      AN    "A 4.4";
      A     "CARR_FREQ_CONV_RUN";
      A(;
      A     "U3_INCREASE_FINE";
      A     "T24_CARR_SPEED_ADJUST";
      O     "U3_INCREASE_COARSE";
      );
      =     "A 4.3";
NETWORK
TITLE =
      AN    "A 4.3";
      A     "CARR_FREQ_CONV_RUN";
      A(;
      A     "U3_REDUSE_FINE";
      A     "T24_CARR_SPEED_ADJUST";
      O     "U3_REDUSE_COARSE";
      );
      =     "A 4.4";
NETWORK
TITLE = CARRIAGE MOTOR STANDS STILL, OK TO START
      L     500;
      L     PIW 754;
      >=I;
      =     "CARR_OK_TO_START";
END_FUNCTION

FUNCTION "TOPPLATE" : VOID	// FC 24
TITLE = TOPPLATE
AUTHOR : LKA
NAME : TOPPLATE
VERSION : 0.1
BEGIN
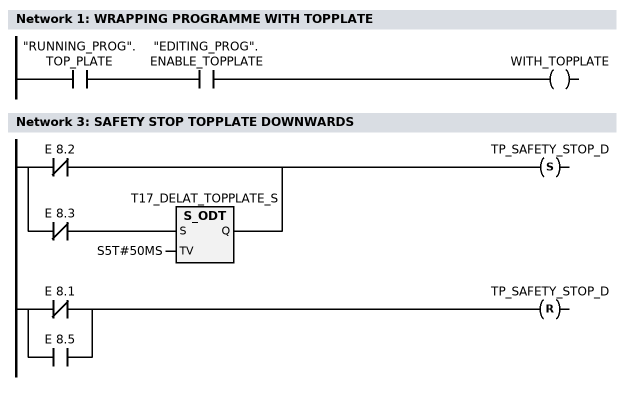
NETWORK
TITLE = WRAPPING PROGRAMME WITH TOPPLATE
      A     "RUNNING_PROG".TOP_PLATE;
      A     "EDITING_PROG".ENABLE_TOPPLATE;
      =     "WITH_TOPPLATE";
NETWORK
TITLE = TOPPLATE UPWARDS
      A(;
      O(;
      A     "HELP_TP_UPWARDS";
      AN    "A 5.6";
      R     "HELP_TP_UPWARDS";
      A(;
      O(;
      A     "RESET_STEP5";
      S     M 90.7;
      AN    "E 8.1";
      R     M 90.7;
      A     M 90.7;
      );
      O     "ST.FC12";
      O(;
      A     "E 124.3";
      FP    M 98.6;
      A     "MACHINE_OK_TO_START";
      );
      O;
      A(;
      L     "RUNNING_PROG".CNT_PULSES_ACT_WRAP;
      L     40;
      >=I;
      );
      A(;
      O     "ST.FC10";
      O     "ST.FC11";
      );
      A     "AUTO";
      A     "EDITING_PROG".OUT_90;
      );
      S     "HELP_TP_UPWARDS";
      A     "HELP_TP_UPWARDS";
      );
      O;
      A     "OK_RUN_BY_HAND";
      A     "E 8.5";
      );
      A     "E 8.1";
      A     "MACHINE__STOP";
      =     "A 5.6";
NETWORK
TITLE = SAFETY STOP TOPPLATE DOWNWARDS
      A(;
      ON    "E 8.2";
      O(;
      AN    "E 8.3";
      L     S5T#50MS;
      SD    "T17_DELAT_TOPPLATE_S";
      NOP   0;
      NOP   0;
      NOP   0;
      A     "T17_DELAT_TOPPLATE_S";
      );
      );
      S     "TP_SAFETY_STOP_D";
      A(;
      ON    "E 8.1";
      O     "E 8.5";
      );
      R     "TP_SAFETY_STOP_D";
      NOP   0;
NETWORK
TITLE = K55 TOPPLATE DOWNWARDS
      O(;
      A     "ST.FC1";
      A     "WITH_TOPPLATE";
      AN    "TP_SAFETY_STOP_D";
      S     "HELP_TP_DOWNWARDS";
      A(;
      O     "TP_SAFETY_STOP_D";
      ON    "MACHINE__STOP";
      O     "E 124.3";
      );
      R     "HELP_TP_DOWNWARDS";
      A     "HELP_TP_DOWNWARDS";
      );
      O;
      A     "OK_RUN_BY_HAND";
      A     "E 8.6";
      AN    "TP_SAFETY_STOP_D";
      =     "A 5.7";
END_FUNCTION

FUNCTION "FILM_FEED_SYSTEM" : VOID	// FC 25
TITLE = FILM FEED SYSTEM
AUTHOR : LKA
NAME : FILMFEED
VERSION : 0.1
BEGIN
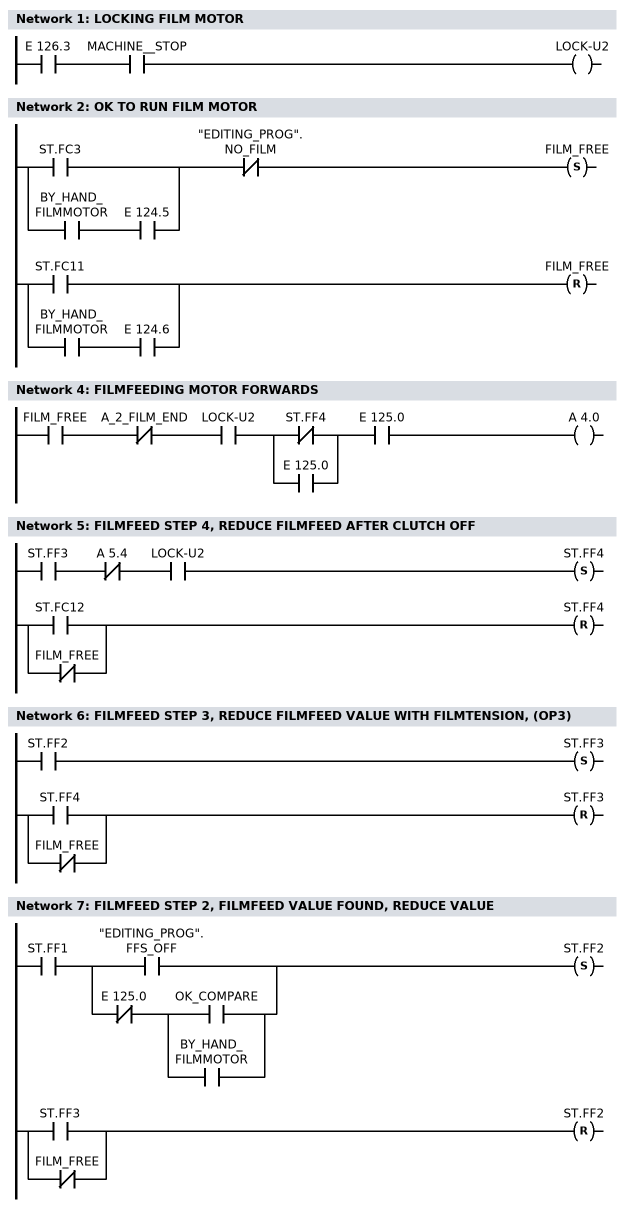
NETWORK
TITLE = LOCKING FILM MOTOR
      A     "E 126.3";
      A     "MACHINE__STOP";
      =     "LOCK-U2";
NETWORK
TITLE = OK TO RUN FILM MOTOR
      A(;
      O     "ST.FC3";
      O;
      A     "BY_HAND_FILMMOTOR";
      A     "E 124.5";
      );
      AN    "EDITING_PROG".NO_FILM;
      S     "FILM_FREE";
      A(;
      O     "ST.FC11";
      O;
      A     "BY_HAND_FILMMOTOR";
      A     "E 124.6";
      );
      R     "FILM_FREE";
      NOP   0;
NETWORK
TITLE = CLUTCH ON
//EV TIDIGARE ÄN ST.FC13
      A(;
      O     "FILM_FREE";
      O(;
      A     "ST.FC13";
      A     "E 125.7";
      S     "CLUTCH_ON_CUT";
      A     "ST.FC16";
      R     "CLUTCH_ON_CUT";
      A     "CLUTCH_ON_CUT";
      );
      );
      AN    "CLUTCH_OFF";
      AN    "ST.FC11";
      A     "LOCK-U2";
      AN    "EDITING_PROG".NO_FILM;
      =     "A 5.4";
NETWORK
TITLE = FILMFEEDING MOTOR FORWARDS
      A     "FILM_FREE";
      AN    "A_2_FILM_END";
      A     "LOCK-U2";
      A(;
      ON    "ST.FF4";
      O     "E 125.0";
      );
      A     "E 125.0";
      =     "A 4.0";
NETWORK
TITLE = FILMFEED STEP 4, REDUCE FILMFEED AFTER CLUTCH OFF
//Minska börvärde efter koppling från.
      A     "ST.FF3";
      AN    "A 5.4";
      A     "LOCK-U2";
      S     "ST.FF4";
      A(;
      O     "ST.FC12";
      ON    "FILM_FREE";
      );
      R     "ST.FF4";
      NOP   0;
NETWORK
TITLE = FILMFEED STEP 3, REDUCE FILMFEED VALUE WITH FILMTENSION, (OP3)
//Hittat 100 % filmutmatning klart, minska med display värde och kör.
      A     "ST.FF2";
      S     "ST.FF3";
      A(;
      O     "ST.FF4";
      ON    "FILM_FREE";
      );
      R     "ST.FF3";
      NOP   0;
NETWORK
TITLE = FILMFEED STEP 2, FILMFEED VALUE FOUND, REDUCE VALUE
//Minska upp mätt analovärde med X %
//
      A     "ST.FF1";
      A(;
      O     "EDITING_PROG".FFS_OFF;
      O;
      AN    "E 125.0";
      A(;
      O     "OK_COMPARE";
      O     "BY_HAND_FILMMOTOR";
      );
      );
      S     "ST.FF2";
      A(;
      O     "ST.FF3";
      ON    "FILM_FREE";
      );
      R     "ST.FF2";
      NOP   0;
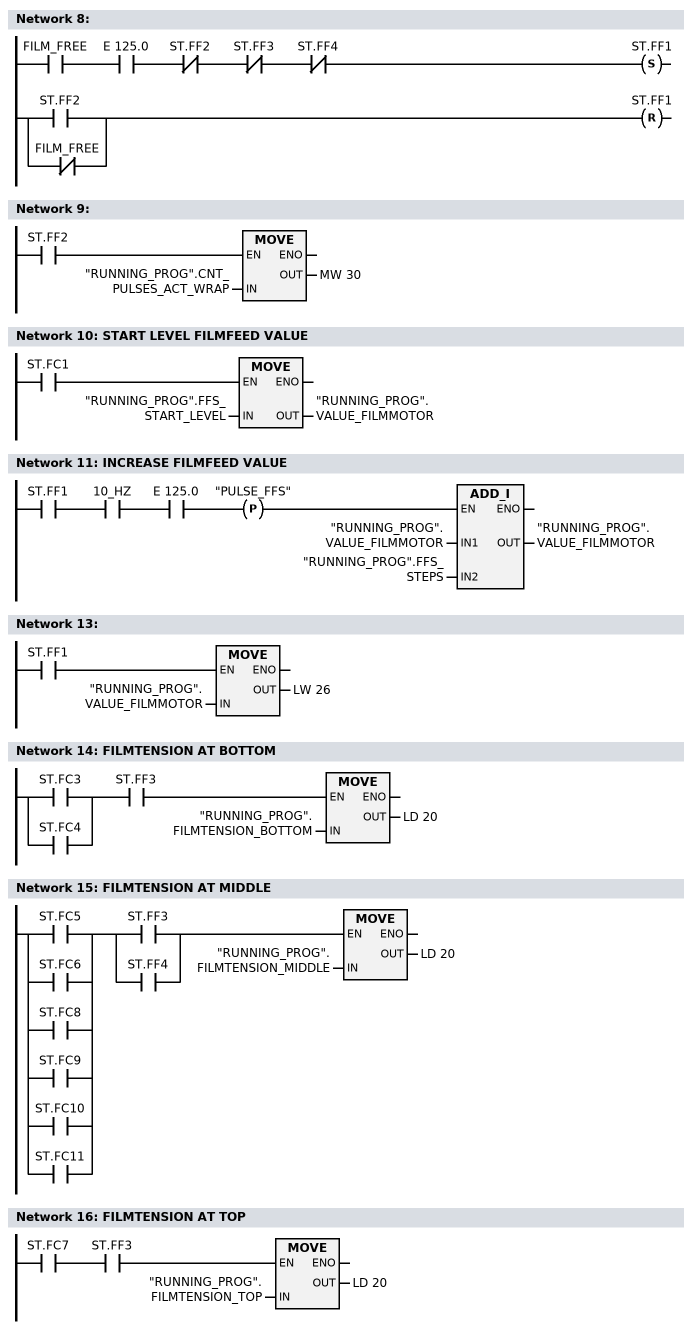
NETWORK
TITLE =
//Rampa upp analogvärde till filmmotor
      A     "FILM_FREE";
      A     "E 125.0";
      AN    "ST.FF2";
      AN    "ST.FF3";
      AN    "ST.FF4";
      S     "ST.FF1";
      A(;
      O     "ST.FF2";
      ON    "FILM_FREE";
      );
      R     "ST.FF1";
      NOP   0;
NETWORK
TITLE =
//denna skall efter test bort!!!!!!!!!!!
//!!!!!!!!!!!!!!!!!!!!!!!!!!!!!!!!!!!!!!
      A     "ST.FF2";
      JNB   _001;
      L     "RUNNING_PROG".CNT_PULSES_ACT_WRAP;
      T     MW 30;
_001: NOP   0;
NETWORK
TITLE = START LEVEL FILMFEED VALUE
//start värde före ändring 2000
      A     "ST.FC1";
      JNB   _002;
      L     "RUNNING_PROG".FFS_START_LEVEL;
      T     "RUNNING_PROG".VALUE_FILMMOTOR;
_002: NOP   0;
NETWORK
TITLE = INCREASE FILMFEED VALUE
//Kolla om väret är rätt, snabbare eller långsammare ramp, (200)
      A     "ST.FF1";
      A     "10_HZ";
      A     "E 125.0";
      FP    "PULSE_FFS";
      JNB   _003;
      L     "RUNNING_PROG".VALUE_FILMMOTOR;
      L     "RUNNING_PROG".FFS_STEPS;
      +I;
      T     "RUNNING_PROG".VALUE_FILMMOTOR;
_003: NOP   0;
NETWORK
TITLE = REDUCE FILMFEED VALUE
//Minska hittat värde med 33 %?? kollas, ev justerbart via display
//Första L#100 var 75!åter!
      A     "ST.FF2";
      AN    "EDITING_PROG".FFS_OFF;
      JCN   M001;
      L     "RUNNING_PROG".VALUE_FILMMOTOR;
      T     MW 200;
      ITD;
      L     L#75;
      *D;
      L     L#100;
      /D;
      T     LD 8;
      L     LW 10;
      T     "RUNNING_PROG".VALUE_FILMMOTOR;
M001: NOP   0;
NETWORK
TITLE =
      A     "ST.FF1";
      JNB   _004;
      L     "RUNNING_PROG".VALUE_FILMMOTOR;
      T     LW 26;
_004: NOP   0;
NETWORK
TITLE = FILMTENSION AT BOTTOM
      A(;
      O     "ST.FC3";
      O     "ST.FC4";
      );
      A     "ST.FF3";
      JNB   _005;
      L     "RUNNING_PROG".FILMTENSION_BOTTOM;
      T     LD 20;
_005: NOP   0;
NETWORK
TITLE = FILMTENSION AT MIDDLE
      A(;
      O     "ST.FC5";
      O     "ST.FC6";
      O     "ST.FC8";
      O     "ST.FC9";
      O     "ST.FC10";
      O     "ST.FC11";
      );
      A(;
      O     "ST.FF3";
      O     "ST.FF4";
      );
      JNB   _006;
      L     "RUNNING_PROG".FILMTENSION_MIDDLE;
      T     LD 20;
_006: NOP   0;
NETWORK
TITLE = FILMTENSION AT TOP
      A     "ST.FC7";
      A     "ST.FF3";
      JNB   _007;
      L     "RUNNING_PROG".FILMTENSION_TOP;
      T     LD 20;
_007: NOP   0;
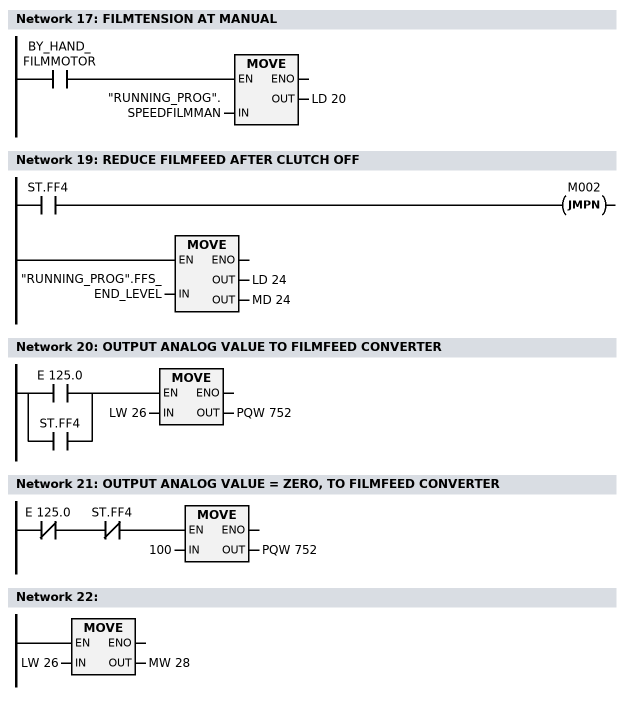
NETWORK
TITLE = FILMTENSION AT MANUAL
      A     "BY_HAND_FILMMOTOR";
      JNB   _008;
      L     "RUNNING_PROG".SPEEDFILMMAN;
      T     LD 20;
_008: NOP   0;
NETWORK
TITLE = REDUCE FILMFEED WITH FILM TENSION
//MINSKA MED FILMSPÄNNINGEN
//MD 24 BORT!!!!!!!!!!!!!!!!!!!!!!
      A     "ST.FF3";
      O     "ST.FF4";
      JCN   M003;
      L     1.000000e+02;
      L     LD 20;
      DTR;
      -R;
      L     "RUNNING_PROG".VALUE_FILMMOTOR;
      ITD;
      DTR;
      *R;
      L     1.000000e+02;
      /R;
      RND;
      T     LD 24;
      T     MD 24;
M003: NOP   0;
NETWORK
TITLE = REDUCE FILMFEED AFTER CLUTCH OFF
//MD 24 BORT!!!!!!!!!!!!!!!!!!!!!!
      A     "ST.FF4";
      JCN   M002;
      L     "RUNNING_PROG".FFS_END_LEVEL;
      T     LD 24;
// temp för visning
      T     MD 24;
M002: NOP   0;
NETWORK
TITLE = OUTPUT ANALOG VALUE TO FILMFEED CONVERTER
      A(;
      O     "E 125.0";
      O     "ST.FF4";
      );
      JNB   _009;
      L     LW 26;
      T     PQW 752;
_009: NOP   0;
NETWORK
TITLE = OUTPUT ANALOG VALUE = ZERO, TO FILMFEED CONVERTER
      AN    "E 125.0";
      AN    "ST.FF4";
      JNB   _00a;
      L     100;
      T     PQW 752;
_00a: NOP   0;
NETWORK
TITLE =
//skall bort!!!!!!
      L     LW 26;
      T     MW 28;
      NOP   0;
END_FUNCTION

FUNCTION "FILM_HOLDING_DEVICE" : VOID	// FC 26
TITLE = FILM HOLDER DEVICE
AUTHOR : LKA
NAME : FILMHOLD
VERSION : 0.0
BEGIN
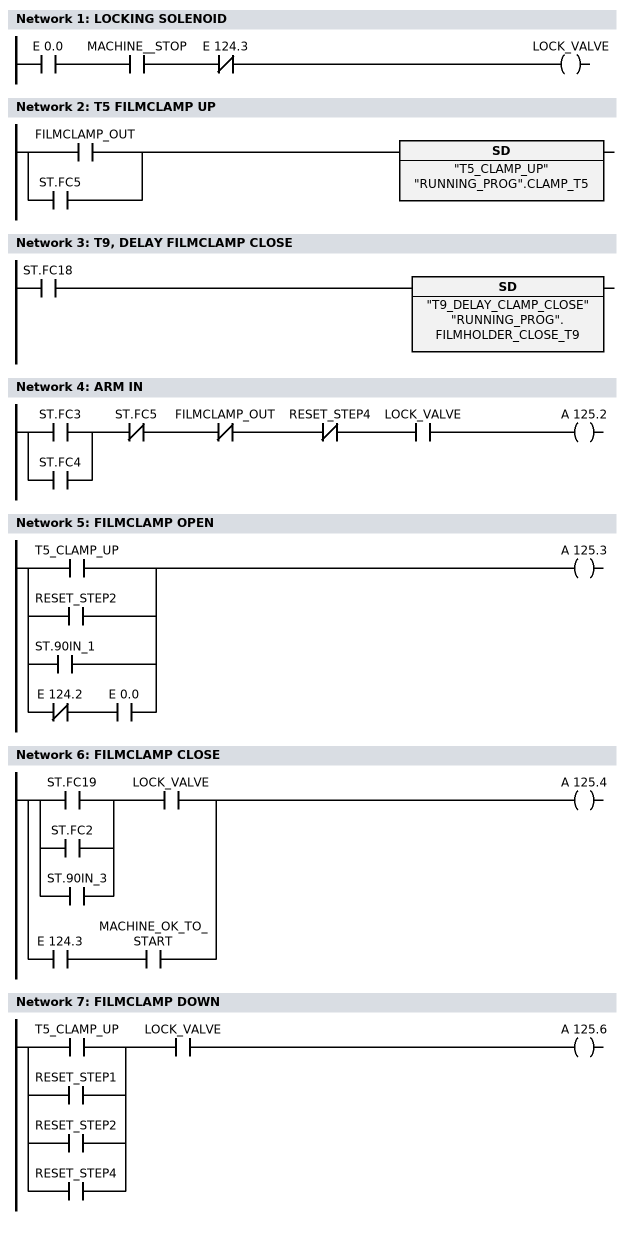
NETWORK
TITLE = LOCKING SOLENOID
      A     "E 0.0";
      A     "MACHINE__STOP";
      AN    "E 124.3";
      =     "LOCK_VALVE";
NETWORK
TITLE = T5 FILMCLAMP UP
      O     "FILMCLAMP_OUT";
      O     "ST.FC5";
      L     "RUNNING_PROG".CLAMP_T5;
      SD    "T5_CLAMP_UP";
NETWORK
TITLE = T9, DELAY FILMCLAMP CLOSE
      A     "ST.FC18";
      L     "RUNNING_PROG".FILMHOLDER_CLOSE_T9;
      SD    "T9_DELAY_CLAMP_CLOSE";
NETWORK
TITLE = ARM IN
      A(;
      O     "ST.FC3";
      O     "ST.FC4";
      );
      AN    "ST.FC5";
      AN    "FILMCLAMP_OUT";
      AN    "RESET_STEP4";
      A     "LOCK_VALVE";
      =     "A 125.2";
NETWORK
TITLE = FILMCLAMP OPEN
      O     "T5_CLAMP_UP";
      O     "RESET_STEP2";
      O     "ST.90IN_1";
      O;
      AN    "E 124.2";
      A     "E 0.0";
      =     "A 125.3";
NETWORK
TITLE = FILMCLAMP CLOSE
      A(;
      O     "ST.FC19";
      O     "ST.FC2";
      O     "ST.90IN_3";
      );
      A     "LOCK_VALVE";
      O;
      A     "E 124.3";
      A     "MACHINE_OK_TO_START";
      =     "A 125.4";
NETWORK
TITLE = FILMCLAMP DOWN
//????????? 3 STEG TILL UTGÅNGSLÄGE ?????????
      A(;
      O     "T5_CLAMP_UP";
      O     "RESET_STEP1";
      O     "RESET_STEP2";
      O     "RESET_STEP4";
      );
      A     "LOCK_VALVE";
      =     "A 125.6";
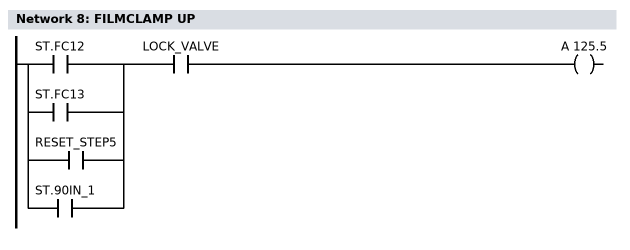
NETWORK
TITLE = FILMCLAMP UP
      A(;
      O     "ST.FC12";
      O     "ST.FC13";
      O     "RESET_STEP5";
      O     "ST.90IN_1";
      );
      A     "LOCK_VALVE";
      =     "A 125.5";
END_FUNCTION

FUNCTION "CUTTING_UNIT" : VOID	// FC 27
TITLE = CUTTING UNIT
AUTHOR : LKA
NAME : CUT_UNIT
VERSION : 0.0
BEGIN
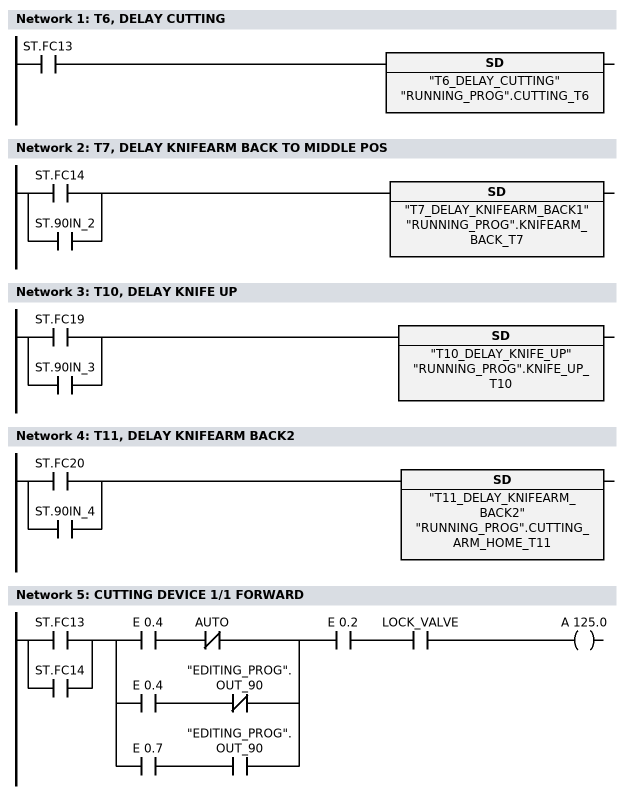
NETWORK
TITLE = T6, DELAY CUTTING
      A     "ST.FC13";
      L     "RUNNING_PROG".CUTTING_T6;
      SD    "T6_DELAY_CUTTING";
NETWORK
TITLE = T7, DELAY KNIFEARM BACK TO MIDDLE POS
      O     "ST.FC14";
      O     "ST.90IN_2";
      L     "RUNNING_PROG".KNIFEARM_BACK_T7;
      SD    "T7_DELAY_KNIFEARM_BACK1";
NETWORK
TITLE = T10, DELAY KNIFE UP
      O     "ST.FC19";
      O     "ST.90IN_3";
      L     "RUNNING_PROG".KNIFE_UP_T10;
      SD    "T10_DELAY_KNIFE_UP";
NETWORK
TITLE = T11, DELAY KNIFEARM BACK2
      O     "ST.FC20";
      O     "ST.90IN_4";
      L     "RUNNING_PROG".CUTTING_ARM_HOME_T11;
      SD    "T11_DELAY_KNIFEARM_BACK2";
NETWORK
TITLE = CUTTING DEVICE 1/1 FORWARD
      A(;
      O     "ST.FC13";
      O     "ST.FC14";
      );
      A(;
      A     "E 0.4";
      AN    "AUTO";
      O;
      A     "E 0.4";
      AN    "EDITING_PROG".OUT_90;
      O;
      A     "E 0.7";
      A     "EDITING_PROG".OUT_90;
      );
      A     "E 0.2";
      A     "LOCK_VALVE";
      =     "A 125.0";
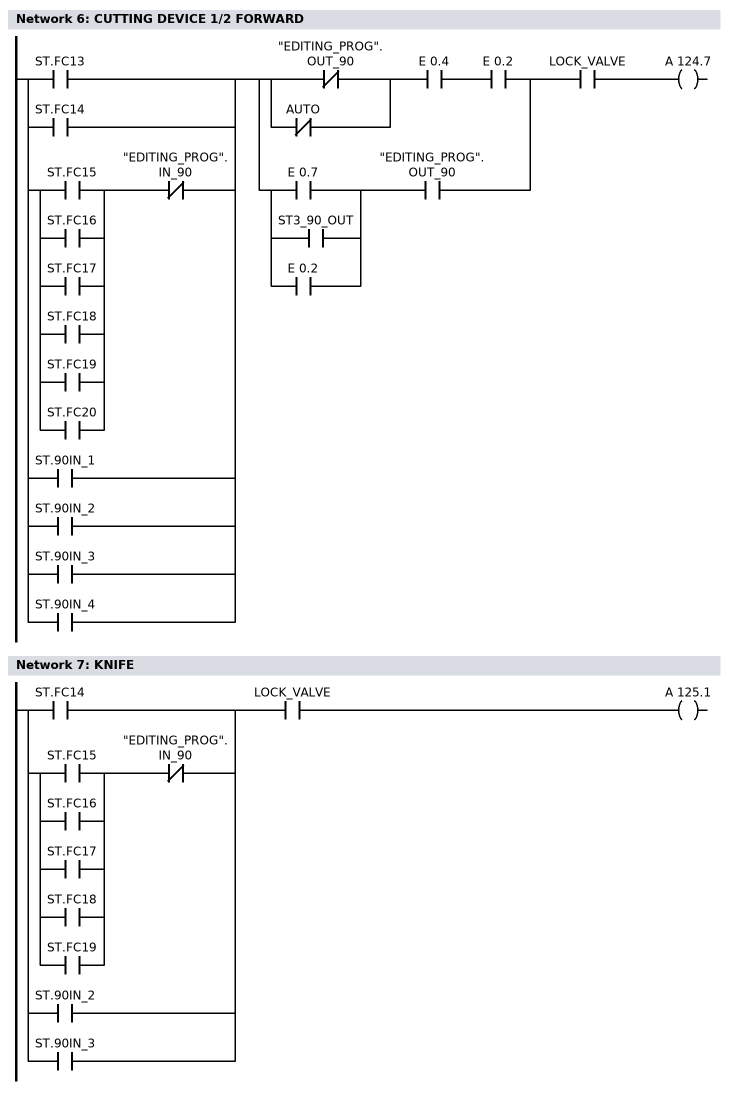
NETWORK
TITLE = CUTTING DEVICE 1/2 FORWARD
//S/R VIPPA ? !!!!!!!!!!!!!!!!!!!!!
      A(;
      O     "ST.FC13";
      O     "ST.FC14";
      O;
      A(;
      O     "ST.FC15";
      O     "ST.FC16";
      O     "ST.FC17";
      O     "ST.FC18";
      O     "ST.FC19";
      O     "ST.FC20";
      );
      AN    "EDITING_PROG".IN_90;
      O     "ST.90IN_1";
      O     "ST.90IN_2";
      O     "ST.90IN_3";
      O     "ST.90IN_4";
      );
      A(;
      A(;
      ON    "EDITING_PROG".OUT_90;
      ON    "AUTO";
      );
      A     "E 0.4";
      A     "E 0.2";
      O;
      A(;
      O     "E 0.7";
      O     "ST3_90_OUT";
      O     "E 0.2";
      );
      A     "EDITING_PROG".OUT_90;
      );
      A     "LOCK_VALVE";
      =     "A 124.7";
NETWORK
TITLE = KNIFE
      A(;
      O     "ST.FC14";
      O;
      A(;
      O     "ST.FC15";
      O     "ST.FC16";
      O     "ST.FC17";
      O     "ST.FC18";
      O     "ST.FC19";
      );
      AN    "EDITING_PROG".IN_90;
      O     "ST.90IN_2";
      O     "ST.90IN_3";
      );
      A     "LOCK_VALVE";
      =     "A 125.1";
END_FUNCTION

FUNCTION "HOT_AIR_WELDING" : VOID	// FC 28
TITLE = HOT AIR WELDING, OPTION
//Folie am Paket ansiegeln, OPTION
//Bausteinaufgaben:
//Dieser Baustein steuert das Ansiegelsystem am  Folienschlitten des Wicklers.
//Hier sind enthalten, Verriegelung, einschalten der Heizung und der Druckluft 
//für die Heizgebläse und Bildung der Schweißzeit.
VERSION : 0.0
BEGIN
